(* Schneider Machine Expert - Basic project Garage_Door, file version 3.0.0.0 *)
(* ProjectInformations: Name=Garage_Door *)

HARDWARE
  Cpu 0: TM221CE24T
  EthernetConfiguration: NetworkName=M221, IpAllocationMode=ByDhcp, IpAddress=192.168.1.10, SubnetMask=255.255.255.0
  SerialLineConfiguration: Baud=Baud19200, Parity=ParityEven, DataBits=DataBits8, StopBits=StopBits1, PhysicalMedium=PhysicalMediumRs485, TransmissionMode=TransmissionModeModbusRtu, SlaveId=1, Addressing=SlaveAddressing
  MastTask: UsePeriodScanMode=false, PeriodScan=100
  FastTask: Period=255
  CpuBehavior: StartingMode=StartAsPreviousState, AutoSaveRamOnEeprom=true, WatchdogPeriod=250

SYMBOLS  (address, symbol, comment, settings)
  %M0       MTR_UP_RUN  "motor UP relay state"
  %M1       MTR_DOWN_RUN  "motor DOWN relay state"
  %I0.1     PB_UP
  %I0.2     PB_DOWN
  %I0.3     LS_UPPER
  %I0.4     LS_LOWER
  %Q0.0     MTR_UP
  %Q0.1     MTR_DOWN

POU Garage_Door
  (* SectionNumber=1 *)

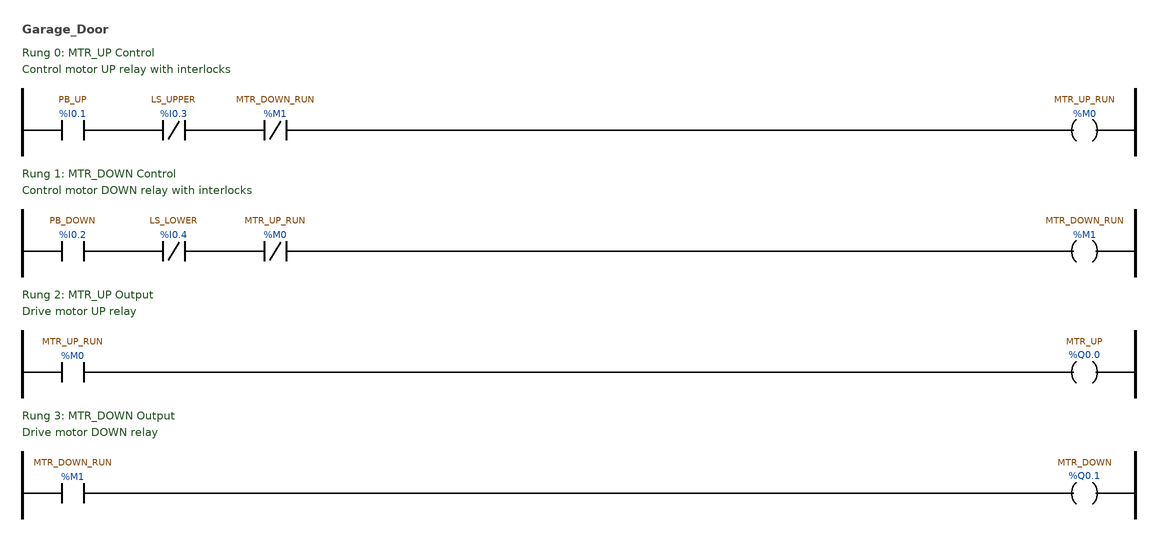

// Rung 0: MTR_UP Control
// Control motor UP relay with interlocks
  LD %I0.1                (* PB_UP *)
  ANDN %I0.3              (* LS_UPPER *)
  ANDN %M1                (* MTR_DOWN_RUN *)
  ST %M0                  (* MTR_UP_RUN *)
  // as ST:
  //   MTR_UP_RUN := PB_UP AND NOT LS_UPPER AND NOT MTR_DOWN_RUN;

// Rung 1: MTR_DOWN Control
// Control motor DOWN relay with interlocks
  LD %I0.2                (* PB_DOWN *)
  ANDN %I0.4              (* LS_LOWER *)
  ANDN %M0                (* MTR_UP_RUN *)
  ST %M1                  (* MTR_DOWN_RUN *)
  // as ST:
  //   MTR_DOWN_RUN := PB_DOWN AND NOT LS_LOWER AND NOT MTR_UP_RUN;

// Rung 2: MTR_UP Output
// Drive motor UP relay
  LD %M0                  (* MTR_UP_RUN *)
  ST %Q0.0                (* MTR_UP *)
  // as ST:
  //   MTR_UP := MTR_UP_RUN;

// Rung 3: MTR_DOWN Output
// Drive motor DOWN relay
  LD %M1                  (* MTR_DOWN_RUN *)
  ST %Q0.1                (* MTR_DOWN *)
  // as ST:
  //   MTR_DOWN := MTR_DOWN_RUN;
